{attribute 'GeneratedUsingTerminal: EL6201-0000-0017'}
{attribute addProperty BoxType "EL6201-0000-0017"}
{attribute addProperty Id "Slave_9A_DO0BOOL1Slave_9A_DO1BOOL1Slave_9A_DO2BOOL1Slave_9A_DO3BOOL1Slave_9B_DO0BOOL1Slave_9B_DO1BOOL1Slave_9B_DO2BOOL1Slave_9B_DO3BOOL1"}
{attribute addProperty CRC "1566342343"}
{attribute addProperty Size "8"}
TYPE Slave_9_Outputs_5D5C7CC7 :
STRUCT
	{attribute addProperty Name "Slave_9A_DO0"}
	Slave_9A_DO0 : BOOL;
	{attribute addProperty Name "Slave_9A_DO1"}
	Slave_9A_DO1 : BOOL;
	{attribute addProperty Name "Slave_9A_DO2"}
	Slave_9A_DO2 : BOOL;
	{attribute addProperty Name "Slave_9A_DO3"}
	Slave_9A_DO3 : BOOL;
	{attribute addProperty Name "Slave_9B_DO0"}
	Slave_9B_DO0 : BOOL;
	{attribute addProperty Name "Slave_9B_DO1"}
	Slave_9B_DO1 : BOOL;
	{attribute addProperty Name "Slave_9B_DO2"}
	Slave_9B_DO2 : BOOL;
	{attribute addProperty Name "Slave_9B_DO3"}
	Slave_9B_DO3 : BOOL;
END_STRUCT
END_TYPE

(* stored: Version 1.2.0.0, ProductVersion 3.1.4024.9
   DUT Slave_9_Outputs_5D5C7CC7: Id {cdf3d1ad-e61c-4857-b4f0-589e0f42fe5a} *)
